TYPE ChuckConfigs :
STRUCT
	PsdChuckConfig : PsdChuckConfig;
	PhotoLumChuckConfig : PhotoLumChuckConfig;
END_STRUCT
END_TYPE

(* stored: Version 1.1.0.1, ProductVersion 3.1.4024.12
   DUT ChuckConfigs: Id {22341ea6-66e6-487a-9d3b-b6ab91005bc4} *)
